// TIA Portal V19 export
FUNCTION "FC_KorrPos" : Void   // FC216, STL
{ S7_Optimized_Access := 'FALSE' }
// stored: AutoNumber false
   VAR_INPUT
      TW_Nr : Int;   // Fahrwagennummer
      IstPos : Byte;   // Istposition aus Messbaustein
      ErrCount : Byte;   // Messwert ungültig bei <>0
      Laser_on : Bool;   // Messwert neu --> Korrektur
   END_VAR
   VAR_IN_OUT
      PosInc : DInt;   // IstPosition TW
   END_VAR
   VAR_TEMP
      IstPosInc : DInt;
      CheckPosInc : DInt;
      Korrektur : DInt;
      CheckPosKorr : DInt;
      s_max : Real;   // Abstand zwischen den Pos.
      s_ist : Real;   // Abstand zur Istposition
      KorrDiff : Real;   // Differenz beider Korrekturwerte
      CheckPos : Int;
      FW_DB : Int;
   END_VAR
BEGIN

NETWORK
TITLE = Initialisieren
//Korrekturrechnung deaktiviert
      AN    "DB_KorrPos".Berechnung_ein;
      O     "DB_ANLAGE".BA.Mess_on;
      BEC;

//erster Durchlauf ohne Korrektur
      L     #IstPos;
      L     0;
      ==I;
      BEC;

//Messsystem liefert gerade keinen Messwert
      L     #ErrCount;
      L     0;
      <>I;
      ON    #Laser_on;
      BEC;


NETWORK
TITLE = Inkremente holen Istposition
      L     #IstPos;
      L     "DB_POS".LENG;
      *D;
      L     "DB_POS".Offset;
      +D;
      SLD   3;
      LAR1;
      OPN   "DB_POS";
      L     DBD [AR1, P#22.0];  //"DB_POS".POS[0].IncPos
      T     #IstPosInc;

      L     #TW_Nr;
      +     -1;
      L     "DB_KorrPos".Leng;
      *D;
      L     "DB_KorrPos".Offset;
      +D;
      SLD   3;
      LAR1;  //Adresse Start TWx
      OPN   "DB_KorrPos";
      L     #IstPos;
      +     -1;
      L     2;
      *D;
      SLD   3;
      +AR1;  //Adresse Posy zu TWx
      L     DBW [AR1, P#0.0];  //"DB_KorrPos".TW1[1].Pos[1]
      ITD;
      NEGD;  //Invertieren, weil positiver Offset negative Korrektur bedeutet
      T     #Korrektur;

      L     #PosInc;
      L     #IstPosInc;
      -D;
//höhere Pos testen
      JP    hPos;
//niedrigere Pos testen
      JM    nPos;
//genau mittig
      JU    Out;

//Höhere Position Testen
hPos: L     "DB_ANLAGE".config.ANZ_Pos;  //Es existiert keine größere Pos.
      L     #IstPos;
      <=I;
      JC    Out;
      +     1;
      T     #CheckPos;
      JU    Chk;

//Niedrigere Position Testen
nPos: L     1;  //Es existiert keine niedrigere Pos.
      L     #IstPos;
      >=I;
      JC    Out;
      +     -1;
      T     #CheckPos;
      JU    Chk;


NETWORK
TITLE = Checkposdaten holen
Chk:  L     #CheckPos;
      L     "DB_POS".LENG;
      *D;
      L     "DB_POS".Offset;
      +D;
      SLD   3;
      LAR1;
      OPN   "DB_POS";
      L     DBD [AR1, P#22.0];  //"DB_POS".POS[0].IncPos
      T     #CheckPosInc;

      L     #TW_Nr;
      +     -1;
      L     "DB_KorrPos".Leng;
      *D;
      L     "DB_KorrPos".Offset;
      +D;
      SLD   3;
      LAR1;  //Adresse Start TWx
      OPN   "DB_KorrPos";
      L     #CheckPos;
      +     -1;
      L     2;
      *D;
      SLD   3;
      +AR1;  //Adresse Posy zu TWx
      L     DBW [AR1, P#0.0];  //"DB_KorrPos".TW1[1].Pos[1]
      ITD;
      NEGD;  //Invertieren, weil positiver Offset negative Korrektur bedeutet
      T     #CheckPosKorr;


NETWORK
TITLE = Korrektur berechnen
      L     #IstPosInc;
      L     #Korrektur;
      -D;
      T     #IstPosInc;

      L     #CheckPosInc;
      L     #CheckPosKorr;
      -D;
      T     #CheckPosInc;

      L     #IstPosInc;
      L     #CheckPosInc;
      -D;
      DTR;
      ABS;
      T     #s_max;
      L     0.0;  //Div durch Null (beide Pos gleiches Inc)
      ==R;
      JC    Out;

      L     #IstPosInc;
      L     #PosInc;
      -D;
      DTR;
      ABS;
      T     #s_ist;

      L     #CheckPosKorr;
      L     #Korrektur;
      -D;
      DTR;
      T     #KorrDiff;

      L     #s_ist;
      L     #s_max;
      /R;
      L     #KorrDiff;
      *R;
      RND;
      L     #Korrektur;
      +D;
      T     #Korrektur;


NETWORK
TITLE = Ausgabe
Out:  L     #Korrektur;
      L     #PosInc;
      +D;
      T     #PosInc;

END_FUNCTION
